(* IEC 61131-3 sources: POMIRTS_lab3/AS/Library_2/AsIORTI, 3 files *)

(* ---- AsIORTI.typ ---- *)
TYPE
	IORTI_DOUTTIME : 	STRUCT
		MODE_INACT : UDINT := 16#00000000; (*Digital Output Mode inactiv*)
		MODE_BOOL : UDINT := 16#00000001; (*Digital Output Mode boolean *)
		MODE_BASE_OFFS : UDINT := 16#00000002; (*Digital Output Mode Base and Offset one shot*)
		MODE_BASE_OFFS_PER : UDINT := 16#00000004; (*Digital Output Mode Base and Offset periodic*)
		MODE_ABSOLUT : UDINT := 16#00000008; (*Digital Output Mode absolut comparator values*)
		MODE_BOOL_INV : UDINT := 16#00000011; (*Digital Output Mode boolean inverted*)
		MODE_BASE_OFFS_INV : UDINT := 16#00000012; (*Digital Output Mode Base and Offset one shot  inverted*)
		MODE_BASE_OFFS_PER_INV : UDINT := 16#00000014; (*Digital Output Mode Base and Offset periodic  inverted*)
		MODE_ABSOLUT_INV : UDINT := 16#00000018; (*Digital Output Mode absolut comparator values inverted*)
	END_STRUCT;
	IORTI_COMP : 	STRUCT
		MODE_DISABLE : UDINT := 16#00000000; (*Comp Mode inactive*)
		MODE_ENABLE : UDINT := 16#00000001; (*Comp Mode active*)
		MODE_EQ : UDINT := 16#00000003; (*In1 is equal to In2*)
		MODE_NE : UDINT := 16#0000000D; (*In1 is not equal to In2*)
		MODE_GTU : UDINT := 16#00000005; (*In1 is greater than In2   (unsigned)*)
		MODE_GEU : UDINT := 16#00000007; (*In1 is greater or equal to In2   (unsigned)*)
		MODE_LTU : UDINT := 16#00000009; (*In1 is less than In2   (unsigned)*)
		MODE_LEU : UDINT := 16#0000000B; (*In1 is less or equal to In2   (unsigned)*)
		MODE_GT : UDINT := 16#80000005; (*In1 is greater than In2   (signed)*)
		MODE_GE : UDINT := 16#80000007; (*In1 is greater or equal to In2   (signed)*)
		MODE_LT : UDINT := 16#80000009; (*In1 is less than In2   (signed)*)
		MODE_LE : UDINT := 16#8000000B; (*In1 is less or equal to In2   (signed)*)
	END_STRUCT;
	IORTI_MUL : 	STRUCT
		MODE_UNSIGNED : UDINT := 16#00000000; (*Multiplication Mode unsigned*)
		MODE_SIGNED : UDINT := 16#80000000; (*Multiplication Mode signed*)
	END_STRUCT;
	IORTI_DIV : 	STRUCT
		MODE_UNSIGNED : UDINT := 16#00000000; (*Division Mode unsigned*)
		MODE_SIGNED : UDINT := 16#80000000; (*Division Mode signed*)
	END_STRUCT;
	IORTI_PWM : 	STRUCT
		MODE_INACT : UDINT := 16#00000000; (*Pwm Mode inactiv*)
		MODE_LEFT_PROC : UDINT := 16#00000001; (*Pwm Mode active left aligned  hightime as procentual value*)
		MODE_LEFT_PROC_DB : UDINT := 16#00000009; (*Pwm Mode active left aligned  hightime as procentual value, deadband enable*)
		MODE_LEFT_PROC_INV : UDINT := 16#00000011; (*Pwm Mode active left aligned  hightime as procentual value, inverted*)
		MODE_LEFT_PROC_DB_INV : UDINT := 16#00000019; (*Pwm Mode active left aligned  hightime as procentual value, deadband enable, inverted*)
		MODE_LEFT_TIME : UDINT := 16#00000005; (*Pwm Mode active left aligned  hightime as time value*)
		MODE_LEFT_TIME_DB : UDINT := 16#0000000D; (*Pwm Mode active left aligned  hightime as time value, deadband enable*)
		MODE_LEFT_TIME_INV : UDINT := 16#00000015; (*Pwm Mode active left aligned  hightime as time value, inverted*)
		MODE_LEFT_TIME_DB_INV : UDINT := 16#0000001D; (*Pwm Mode active left aligned  hightime as time value, deadband enable, inverted*)
		MODE_CENT_PROC : UDINT := 16#00000003; (*Pwm Mode active centered hightime as procentual value*)
		MODE_CENT_PROC_DB : UDINT := 16#0000000B; (*Pwm Mode active centered hightime as procentual value, deadband enable*)
		MODE_CENT_PROC_INV : UDINT := 16#00000013; (*Pwm Mode active centered hightime as procentual value, inverted*)
		MODE_CENT_PROC_DB_INV : UDINT := 16#0000001B; (*Pwm Mode active centered hightime as procentual value, deadband enable, inverted*)
		MODE_CENT_TIME : UDINT := 16#00000007; (*Pwm Mode active centered hightime as time value*)
		MODE_CENT_TIME_DB : UDINT := 16#0000000F; (*Pwm Mode active centered hightime as time value, deadband enable*)
		MODE_CENT_TIME_INV : UDINT := 16#00000017; (*Pwm Mode active centered hightime as time value, inverted*)
		MODE_CENT_TIME_DB_INV : UDINT := 16#0000001F; (*Pwm Mode active centered hightime as time value, deadband enable, inverted*)
		MODE_USE_START_AS_BASE : UDINT := 16#00000020; (*Pwm Mode Start used as Basetime*)
	END_STRUCT;
	IORTI_COUNT : 	STRUCT
		MODE_UPDWN_NOSTOP : UDINT := 16#00000000; (*Eventcounter Mode Up/Down with overrun*)
		MODE_CLKDIR_NOSTOP : UDINT := 16#00000001; (*Eventcounter Mode Clock and direction with overrun*)
		MODE_UPDWN_STOP : UDINT := 16#00000002; (*Eventcounter Mode Up/Down, stop at overrun*)
		MODE_CLKDIR_STOP : UDINT := 16#00000003; (*Eventcounter Mode Clock and direction, stop at overrun*)
	END_STRUCT;
	IORTI_REGISTER : 	STRUCT
		MODE_FREEZED : UDINT := 16#00000000; (*Register freezed*)
		MODE_TRANSPARENT : UDINT := 16#00000001; (*Register transparent*)
		MODE_EDGE_RISING : UDINT := 16#00000010; (*Register latch on rising edge*)
		MODE_EDGE_FALLING : UDINT := 16#00000011; (*Register latch on falling edge*)
		MODE_EDGE_BOTH : UDINT := 16#00000012; (*Register latch on both edges*)
		MODE_LEVEL_LOW : UDINT := 16#00000020; (*Register transparent if Latch low*)
		MODE_LEVEL_HIGH : UDINT := 16#00000021; (*Register transparent if Latch high*)
	END_STRUCT;
	IORTI_REAL : 	STRUCT
		TYPE_NORM : DINT := 16#00000000; (*Result is normalized*)
		TYPE_ZERO : DINT := 16#00000001; (*Result is zero*)
		TYPE_NAN : DINT := 16#00000002; (*Result is not a number*)
		TYPE_UNDER : DINT := 16#00000004; (*Result is underflow *)
		TYPE_OVER : DINT := 16#00000008; (*Result is overflow*)
		TYPE_DIVZERO : DINT := 16#00000010; (*Result is divide by zero*)
		TYPE_INFINITE : DINT := 16#00000020; (*Result is infinite*)
	END_STRUCT;
END_TYPE

(* ---- AsIORTI.fun ---- *)
FUNCTION_BLOCK rtiABCnt {ReActionFunctionNr 6}  {ReActionPhysical Channel} {ReActionPhysicalUnique ABR} (*AB Counter with latch*)
	VAR_INPUT
		Channel : INT;
		Mode : DINT;
		LatchEnable : DINT;
		LatchConfig : DINT;
		ForceOn : DINT;
		ForceCnt : DINT;
		ForceLatch : DINT;
		SimulCnt : {ReActionSimulParam} DINT;
		SimulLatch : {ReActionSimulParam} BOOL;
	END_VAR
	VAR_OUTPUT
		Cnt : DINT;
		CntTs : DINT;
		Latch : DINT;
		LatchTs : DINT;
		Status : DINT;
	END_VAR
	VAR
		LocLatch : DINT;
	END_VAR
END_FUNCTION_BLOCK

FUNCTION_BLOCK rtiABRPos {ReActionFunctionNr 7}  {ReActionPhysical Channel} {ReActionPhysicalUnique ABR} (*ABR Counter*)
	VAR_INPUT
		Channel : INT;
		Mode : DINT;
		RefEnable : DINT;
		RefConfig : DINT;
		RefPos : DINT;
		ForceOn : DINT;
		ForceVal : DINT;
		SimulPos : {ReActionSimulParam} DINT;
		SimulRef : {ReActionSimulParam} BOOL;
	END_VAR
	VAR_OUTPUT
		Pos : DINT;
		PosTs : DINT;
		Status : DINT;
	END_VAR
	VAR
		LocRefPos : DINT;
		LocRefDone : DINT;
		LocRefIn : BOOL;
	END_VAR
END_FUNCTION_BLOCK

FUNCTION_BLOCK rtiAbs {ReActionFunctionNr 121}		(*absolute value of signed value*)
	VAR_INPUT
		In : DINT;
	END_VAR
	VAR_OUTPUT
		Out : DINT;
	END_VAR
END_FUNCTION_BLOCK

FUNCTION_BLOCK rtiAdd {ReActionFunctionNr 107}		(*add In1 and In2*)
	VAR_INPUT
		In1 : DINT;
		In2 : DINT;
	END_VAR
	VAR_OUTPUT
		Out : DINT;
	END_VAR
END_FUNCTION_BLOCK

FUNCTION_BLOCK rtiAddSubReal {ReActionFunctionNr 130}	(*add or sub  In1 and In2*)
	VAR_INPUT
		In1 : REAL;
		In2 : REAL;
		Mode : DINT;
	END_VAR
	VAR_OUTPUT
		Out : REAL;
		Status : DINT;
	END_VAR
END_FUNCTION_BLOCK

FUNCTION_BLOCK rtiAin {ReActionFunctionNr 4}  {ReActionPhysical Channel} {ReActionPhysicalUnique}	(*read analog input channel*)
	VAR_INPUT
		Channel : INT;
		Filter : DINT;
		ForceOn : DINT;
		ForceVal : DINT;
		Simul : {ReActionSimulParam} DINT;
	END_VAR
	VAR_OUTPUT
		Out : DINT;
		Status : DINT;
	END_VAR
END_FUNCTION_BLOCK

FUNCTION_BLOCK rtiAnd {ReActionFunctionNr 100}	(*bitwise AND*)
	VAR_INPUT
		In1 : DINT;
		In2 : DINT;
		In3 : DINT;
		In4 : DINT;
	END_VAR
	VAR_OUTPUT
		OutTsEdge : DINT;
		Out : DINT;
		OutN : DINT;
	END_VAR
END_FUNCTION_BLOCK

FUNCTION_BLOCK rtiAnLimit {ReActionFunctionNr 118}	(*limit analog input value*)
	VAR_INPUT
		In : DINT;
		StatusIn : DINT;
		LowLimit : DINT;
		HighLimit : DINT;
	END_VAR
	VAR_OUTPUT
		Out : DINT;
		Status : DINT;
	END_VAR
END_FUNCTION_BLOCK

FUNCTION_BLOCK rtiAout {ReActionFunctionNr 5}  {ReActionPhysical Channel} {ReActionPhysicalUnique} (*write analog output channel*)
	VAR_INPUT
		Channel : INT;
		Enable : DINT;
		In : DINT;
		ForceOn : DINT;
		ForceVal : DINT;
	END_VAR
	VAR_OUTPUT
		OutRef : DINT;
		Simul : {ReActionSimulParam} DINT;
	END_VAR
END_FUNCTION_BLOCK

FUNCTION_BLOCK rtiBit2Byte {ReActionFunctionNr 119}	(*combines 8 bits into 1 byte*)
	VAR_INPUT
		In1 : DINT;
		In2 : DINT;
		In3 : DINT;
		In4 : DINT;
		In5 : DINT;
		In6 : DINT;
		In7 : DINT;
		In8 : DINT;
	END_VAR
	VAR_OUTPUT
		Out : DINT;
	END_VAR
END_FUNCTION_BLOCK

FUNCTION_BLOCK rtiByte2Bit {ReActionFunctionNr 120}	(*splits 1 byte into 8 bits*)
	VAR_INPUT
		In : DINT;
	END_VAR
	VAR_OUTPUT
		Out1 : DINT;
		Out2 : DINT;
		Out3 : DINT;
		Out4 : DINT;
		Out5 : DINT;
		Out6 : DINT;
		Out7 : DINT;
		Out8 : DINT;
	END_VAR
END_FUNCTION_BLOCK

FUNCTION_BLOCK rtiComp {ReActionFunctionNr 104}	(*compares In1 and In2 depending on the Mode*)
	VAR_INPUT
		Mode : UDINT;
		In1 : DINT;
		In2 : DINT;
	END_VAR
	VAR_OUTPUT
		StatusTsEdgePos : DINT;
		Status : DINT;
	END_VAR
END_FUNCTION_BLOCK

FUNCTION_BLOCK rtiCompReal {ReActionFunctionNr 133}	(*compares In1 and In2 depending on the Mode*)
	VAR_INPUT
		Mode : UDINT;
		In1 : REAL;
		In2 : REAL;
	END_VAR
	VAR_OUTPUT
		StatusTsEdgePos : DINT;
		Status : DINT;
		Result : DINT;
	END_VAR
END_FUNCTION_BLOCK

FUNCTION_BLOCK rtiCount {ReActionFunctionNr 115}	(*Up-Down counter or Clock-Direction counter, level sensitive*)
	VAR_INPUT
		Mode : UDINT;
		Up_Clk : DINT;
		Down_Dir : DINT;
		Clear : DINT;
	END_VAR
	VAR_OUTPUT
		OvlTsEdgePos : DINT;
		Out : DINT;
	END_VAR
END_FUNCTION_BLOCK

FUNCTION_BLOCK rtiDelay {ReActionFunctionNr 113}	(*delay signal for 1 reACTION cycle*)
	VAR_INPUT
		In : DINT;
	END_VAR
	VAR_OUTPUT
		Out : DINT;
		Out1 : DINT;
		Out2 : DINT;
		Out3 : DINT;
		Out4 : DINT;
	END_VAR
END_FUNCTION_BLOCK

FUNCTION_BLOCK rtiDelayReal {ReActionFunctionNr 113}	(*delay signal for 1 reACTION cycle*)
	VAR_INPUT
		In : REAL;
	END_VAR
	VAR_OUTPUT
		Out : REAL;
		Out1 : REAL;
		Out2 : REAL;
		Out3 : REAL;
		Out4 : REAL;
	END_VAR
END_FUNCTION_BLOCK

FUNCTION_BLOCK rtiDeMux {ReActionFunctionNr 117}	(*demultiplexer for 4 outputs*)
	VAR_INPUT
		Mux : DINT;
		In : DINT;
	END_VAR
	VAR_OUTPUT
		Out1 : DINT;
		Out2 : DINT;
		Out3 : DINT;
		Out4 : DINT;
	END_VAR
END_FUNCTION_BLOCK

FUNCTION_BLOCK rtiDeMuxReal {ReActionFunctionNr 117}	(*demultiplexer for 4 outputs*)
	VAR_INPUT
		Mux : DINT;
		In : REAL;
	END_VAR
	VAR_OUTPUT
		Out1 : REAL;
		Out2 : REAL;
		Out3 : REAL;
		Out4 : REAL;
	END_VAR
END_FUNCTION_BLOCK

FUNCTION_BLOCK rtiDin {ReActionFunctionNr 1} {ReActionPhysical Channel} {ReActionPhysicalUnique}	(*read digital input channel*)
	VAR_INPUT
		Channel : INT;
		Mode : UDINT;
		Filter : DINT;
		ForceOn : DINT;
		ForceVal : DINT;
		Simul : {ReActionSimulParam} BOOL;
	END_VAR
	VAR_OUTPUT
		OutTsEdgePos : DINT;
		OutTsEdgeNeg : DINT;
		Out : DINT;
	END_VAR
END_FUNCTION_BLOCK

FUNCTION_BLOCK rtiDiv {ReActionFunctionNr 110}	(*division*)
	VAR_INPUT
		Mode : UDINT;
		In1 : DINT;
		In2 : DINT;
	END_VAR
	VAR_OUTPUT
		Quotient : DINT;
		Remainder : DINT;
	END_VAR
END_FUNCTION_BLOCK

FUNCTION_BLOCK rtiDivReal {ReActionFunctionNr 132}	(*division*)
	VAR_INPUT
		In1 : REAL;
		In2 : REAL;
	END_VAR
	VAR_OUTPUT
		Quotient : REAL;
		Status : DINT;
	END_VAR
END_FUNCTION_BLOCK

FUNCTION_BLOCK rtiDout {ReActionFunctionNr 2} {ReActionPhysical Channel}  {ReActionPhysicalUnique DigitalOutputs}	(*write digital output channel*)
	VAR_INPUT
		Channel : INT;
		Enable : DINT;
		In : DINT;
		ForceOn : DINT;
		ForceVal : DINT;
	END_VAR
	VAR_OUTPUT
		Simul : {ReActionSimulParam} BOOL;
	END_VAR
END_FUNCTION_BLOCK

FUNCTION_BLOCK rtiDoutTime {ReActionFunctionNr 3} {ReActionPhysical Channel} {ReActionPhysicalUnique DigitalOutputs}	(*write digital output channel*)
	VAR_INPUT
		Channel : INT;
		Mode : UDINT;
		Comp1 : DINT;
		Comp2 : DINT;
		Base : DINT;
		Period : DINT;
		ForceOn : DINT;
		ForceVal : DINT;
	END_VAR
	VAR_OUTPUT
		EdgeCount : DINT;
		Simul : {ReActionSimulParam} BOOL;
	END_VAR
	VAR
		LocLatch : DINT;
		LocStat : DINT;
	END_VAR
END_FUNCTION_BLOCK

FUNCTION_BLOCK rtiIntToReal {ReActionFunctionNr 128}	 (*convert int to real with decimal point offset*)
	VAR_INPUT
		In : DINT;
		Shift : DINT;
	END_VAR
	VAR_OUTPUT
		Out : REAL;
		Status : DINT;
	END_VAR
END_FUNCTION_BLOCK

FUNCTION_BLOCK rtiInvertReal {ReActionFunctionNr 134}   (*invert input*)
	VAR_INPUT
		In : REAL;
	END_VAR
	VAR_OUTPUT
		Out : REAL;
		Status : DINT;
	END_VAR
END_FUNCTION_BLOCK

FUNCTION_BLOCK rtiLatch {ReActionFunctionNr 105}	(*latch value*)
	VAR_INPUT
		In : DINT;
		Latch : DINT;
	END_VAR
	VAR_OUTPUT
		Out : DINT;
	END_VAR
	VAR
		LocLatch : DINT;
	END_VAR
END_FUNCTION_BLOCK

FUNCTION_BLOCK rtiLatchReal {ReActionFunctionNr 105}	(*latch value*)
	VAR_INPUT
		In : REAL;
		Latch : DINT;
	END_VAR
	VAR_OUTPUT
		Out : REAL;
	END_VAR
END_FUNCTION_BLOCK

FUNCTION_BLOCK rtiMul {ReActionFunctionNr 109}	(*multiplication*)
	VAR_INPUT
		Mode : UDINT;
		In1 : DINT;
		In2 : DINT;
	END_VAR
	VAR_OUTPUT
		OutL : DINT;
		OutH : DINT;
	END_VAR
END_FUNCTION_BLOCK

FUNCTION_BLOCK rtiMulReal {ReActionFunctionNr 131}	(*multiplication*)
	VAR_INPUT
		In1 : REAL;
		In2 : REAL;
	END_VAR
	VAR_OUTPUT
		Out : REAL;
		Status : DINT;
	END_VAR
END_FUNCTION_BLOCK

FUNCTION_BLOCK rtiMux {ReActionFunctionNr 116}	(*select a value from 4 input values*)
	VAR_INPUT
		Mux : DINT;
		In1 : DINT;
		In2 : DINT;
		In3 : DINT;
		In4 : DINT;
	END_VAR
	VAR_OUTPUT
		Out : DINT;
	END_VAR
END_FUNCTION_BLOCK

FUNCTION_BLOCK rtiMuxReal {ReActionFunctionNr 116}	(*select a value from 4 input values*)
	VAR_INPUT
		Mux : DINT;
		In1 : REAL;
		In2 : REAL;
		In3 : REAL;
		In4 : REAL;
	END_VAR
	VAR_OUTPUT
		Out : REAL;
	END_VAR
END_FUNCTION_BLOCK

FUNCTION_BLOCK rtiNot {ReActionFunctionNr 103}	(*bitwise NOT*)
	VAR_INPUT
		In : DINT;
	END_VAR
	VAR_OUTPUT
		Out : DINT;
	END_VAR
END_FUNCTION_BLOCK

FUNCTION_BLOCK rtiOr {ReActionFunctionNr 101}	(*bitwise OR*)
	VAR_INPUT
		In1 : DINT;
		In2 : DINT;
		In3 : DINT;
		In4 : DINT;
	END_VAR
	VAR_OUTPUT
		OutTsEdge : DINT;
		Out : DINT;
		OutN : DINT;
	END_VAR
END_FUNCTION_BLOCK

FUNCTION_BLOCK rtiPar {ReActionPhysical DpNr}	(*read parameter from cyclic datapoint*)
	VAR_INPUT
		DpNr : INT;
		Simul : {ReActionSimulParam} DINT;
	END_VAR
	VAR_OUTPUT
		Data : DINT;
	END_VAR
END_FUNCTION_BLOCK

FUNCTION_BLOCK rtiParReal {ReActionPhysical DpNr}	 (*read parameter from cyclic datapoint*)
	VAR_INPUT
		DpNr : INT;
		Simul : {ReActionSimulParam} REAL;
	END_VAR
	VAR_OUTPUT
		Data : REAL;
	END_VAR
END_FUNCTION_BLOCK

FUNCTION_BLOCK rtiPwm {ReActionFunctionNr 114}	(*generate PWM signal, must be followed by rtiDoutTime*)
	VAR_INPUT
		Mode : UDINT;
		Start : DINT;
		Period : DINT;
		Duty : DINT;
		DeadB : DINT;
	END_VAR
	VAR_OUTPUT
		ModeOut : UDINT;
		OutTsEdgePos : DINT;
		OutTsEdgeNeg : DINT;
		Base : DINT;
		PeriodOut : DINT;
	END_VAR
END_FUNCTION_BLOCK

FUNCTION_BLOCK rtiRealToInt  {ReActionFunctionNr 129}  (*convert real to int with decimal point offset*)
	VAR_INPUT
		In : REAL;
		Shift : DINT;
	END_VAR
	VAR_OUTPUT
		Out : DINT;
		Status : DINT;
	END_VAR
END_FUNCTION_BLOCK

FUNCTION_BLOCK rtiRegister  {ReActionFunctionNr 124} (*register values*)
	VAR_INPUT
		Mode : UDINT;
		Latch : DINT;
		In1 : DINT;
		In2 : DINT;
		In3 : DINT;
		In4 : DINT;
	END_VAR
	VAR_OUTPUT
		OutTsLatch : DINT;
		Out1 : DINT;
		Out2 : DINT;
		Out3 : DINT;
		Out4 : DINT;
	END_VAR
	VAR
		LocLatch : DINT;
	END_VAR
END_FUNCTION_BLOCK

FUNCTION_BLOCK rtiRegisterReal  {ReActionFunctionNr 124} (*register values*)
	VAR_INPUT
		Mode : UDINT;
		Latch : DINT;
		In1 : REAL;
		In2 : REAL;
		In3 : REAL;
		In4 : REAL;
	END_VAR
	VAR_OUTPUT
		OutTsLatch : DINT;
		Out1 : REAL;
		Out2 : REAL;
		Out3 : REAL;
		Out4 : REAL;
	END_VAR
	VAR
		LocLatch : DINT;
	END_VAR
END_FUNCTION_BLOCK

FUNCTION_BLOCK rtiRes {ReActionPhysical DpNr}  {ReActionPhysicalUnique Results}	(*write results to cyclic datapoint*)
	VAR_INPUT
		DpNr : INT;
		Data : DINT;
	END_VAR
	VAR_OUTPUT
		Simul : {ReActionSimulParam} DINT;
	END_VAR
END_FUNCTION_BLOCK

FUNCTION_BLOCK rtiResReal {ReActionPhysical DpNr}  {ReActionPhysicalUnique Results}	(*write results to cyclic datapoint*)
	VAR_INPUT
		DpNr : INT;
		Data : REAL;
	END_VAR
	VAR_OUTPUT
		Simul : {ReActionSimulParam} REAL;
	END_VAR
END_FUNCTION_BLOCK

FUNCTION_BLOCK rtiRF_TRIG {ReActionFunctionNr 122}	(*detect rising/falling edge of input signal*)
	VAR_INPUT
		CLK : DINT;
	END_VAR
	VAR_OUTPUT
		OutEdge : DINT;
		OutEdgePos : DINT;
		OutEdgeNeg : DINT;
	END_VAR
	VAR
		LocLatch : DINT;
	END_VAR
END_FUNCTION_BLOCK

FUNCTION_BLOCK rtiShift {ReActionFunctionNr 111}	(*arithmetic or logigal shift*)
	VAR_INPUT
		In : DINT;
		Shl : DINT;
		Shr : DINT;
	END_VAR
	VAR_OUTPUT
		Out : DINT;
	END_VAR
END_FUNCTION_BLOCK

FUNCTION_BLOCK rtiSineReal {ReActionFunctionNr 136} (*sine*)
	VAR_INPUT
		In : REAL;
	END_VAR
	VAR_OUTPUT
		Out : REAL;
		Status : DINT;
	END_VAR
END_FUNCTION_BLOCK

FUNCTION_BLOCK rtiSqrtReal {ReActionFunctionNr 135}	(*square root*)
	VAR_INPUT
		In : REAL;
	END_VAR
	VAR_OUTPUT
		Out : REAL;
		Status : DINT;
	END_VAR
END_FUNCTION_BLOCK

FUNCTION_BLOCK rtiSRff {ReActionFunctionNr 106}	(*SR flipflop*)
	VAR_INPUT
		InS : DINT;
		InR : DINT;
	END_VAR
	VAR_OUTPUT
		OutTsEdge : DINT;
		Out : DINT;
	END_VAR
END_FUNCTION_BLOCK

FUNCTION_BLOCK rtiSSI {ReActionFunctionNr 8}  {ReActionPhysical Channel} {ReActionPhysicalUnique} (*SSI Encoder*)
	VAR_INPUT
		Channel : INT;
		Mode : DINT;
		Trigger : DINT;
		ForceOn : DINT;
		ForceVal : DINT;
		SimulPos : {ReActionSimulParam} DINT;
	END_VAR
	VAR_OUTPUT
		Pos : DINT;
		PosTs : DINT;
		Status : DINT;
	END_VAR
END_FUNCTION_BLOCK

FUNCTION_BLOCK rtiSub {ReActionFunctionNr 108}	(*subtraction*)
	VAR_INPUT
		In1 : DINT;
		In2 : DINT;
	END_VAR
	VAR_OUTPUT
		Out : DINT;
	END_VAR
END_FUNCTION_BLOCK

FUNCTION_BLOCK rtiTDel {ReActionFunctionNr 112}	(*compare time delays*)
	VAR_INPUT
		Enable : DINT;
		Comp1 : DINT;
		Comp2 : DINT;
		Comp3 : DINT;
		Comp4 : DINT;
		Comp5 : DINT;
		Comp6 : DINT;
		Base : DINT;
	END_VAR
	VAR_OUTPUT
		Out : DINT;
	END_VAR
	VAR
		LocStat : DINT;
	END_VAR
END_FUNCTION_BLOCK

FUNCTION_BLOCK rtiTime {ReActionFunctionNr 252}	(*get time of cycle start and last parameter refresh*)
	VAR_OUTPUT
		TsPar : DINT;
		TsCycle : DINT;
	END_VAR
END_FUNCTION_BLOCK

FUNCTION_BLOCK rtiTimeLoc2Net {ReActionFunctionNr 250}	(*converts local time [10ns] to NetTime [1/256us]*)
	VAR_INPUT
		LocTime : DINT;
	END_VAR
	VAR_OUTPUT
		NetTime : DINT;
	END_VAR
END_FUNCTION_BLOCK

FUNCTION_BLOCK rtiTimeNet2Loc {ReActionFunctionNr 251}	(*converts NetTime [1/256us] to local time [10ns]*)
	VAR_INPUT
		NetTime : DINT;
	END_VAR
	VAR_OUTPUT
		LocTime : DINT;
	END_VAR
END_FUNCTION_BLOCK

FUNCTION_BLOCK rtiTP {ReActionFunctionNr 123}	(*generates TRUE-pulse on rising edge of input signal*)
	VAR_INPUT
		IN : DINT;
		PT : DINT;
	END_VAR
	VAR_OUTPUT
		Q : DINT;
		ET : DINT;
	END_VAR
	VAR
		LocLatch : DINT;
	END_VAR
END_FUNCTION_BLOCK

FUNCTION_BLOCK rtiVarRead {ReActionPhysical DpNr}	(*reads from internal variable*)
	VAR_INPUT
		DpNr : INT;
		Simul : {ReActionSimulParam} DINT;
	END_VAR
	VAR_OUTPUT
		Out : DINT;
	END_VAR
END_FUNCTION_BLOCK

FUNCTION_BLOCK rtiVarReadReal {ReActionPhysical DpNr}	(*reads from internal variable*)
	VAR_INPUT
		DpNr : INT;
		Simul : {ReActionSimulParam} REAL;
	END_VAR
	VAR_OUTPUT
		Out : REAL;
	END_VAR
END_FUNCTION_BLOCK

FUNCTION_BLOCK rtiVarWrite {ReActionPhysical DpNr}  {ReActionPhysicalUnique VarWrite}	(*writes to internal variable*)
	VAR_INPUT
		DpNr : INT;
		In : DINT;
	END_VAR
	VAR_OUTPUT
		Simul : {ReActionSimulParam} DINT;
	END_VAR
END_FUNCTION_BLOCK

FUNCTION_BLOCK rtiVarWriteReal {ReActionPhysical DpNr}  {ReActionPhysicalUnique VarWrite}	(*writes to internal variable*)
	VAR_INPUT
		DpNr : INT;
		In : REAL;
	END_VAR
	VAR_OUTPUT
		Simul : {ReActionSimulParam} REAL;
	END_VAR
END_FUNCTION_BLOCK

FUNCTION_BLOCK rtiXor {ReActionFunctionNr 102}	(*bitwise XOR*)
	VAR_INPUT
		In1 : DINT;
		In2 : DINT;
		In3 : DINT;
		In4 : DINT;
	END_VAR
	VAR_OUTPUT
		OutTsEdge : DINT;
		Out : DINT;
		OutN : DINT;
	END_VAR
END_FUNCTION_BLOCK

FUNCTION_BLOCK rtiSim (*control simulation mode (no effect on reACTION IO module)*)
	VAR_INPUT
		Enable : {ReActionSimulParam} BOOL;
		Mode : {ReActionSimulParam} UDINT;
		Clear : {ReActionSimulParam} BOOL;
	END_VAR
	VAR_OUTPUT
		Cycles : {ReActionSimulParam} UDINT;
		Status : {ReActionSimulParam} UINT;
	END_VAR
END_FUNCTION_BLOCK

(* ---- AsIORTI.var ---- *)
VAR CONSTANT
	IORTI_SIM_MODE_DEFAULT : UDINT := 16#00000001; (* Default simulation mode *)
	IORTI_SIM_ERR_UNKNOWN_MODE : UDINT := 37910; (* unknown simulation mode selected *)
	IORTI_SIM_ERR_OUT_OF_MEMORY : UDINT := 37911; (* out of memory error *)
	IORTI_SIM_ERR_INVALID_DPNR : UDINT := 37912; (* invalid datapoint number *)
	IORTI_SIM_ERR_PAR_SIMUL_VALUE : UDINT := 37913; (* simulation values for parameters with the same DpNr are not equal *)
	IORTI_SIM_ERR_VAR_SIMUL_VALUE : UDINT := 37914; (* simulation values for variables with the same DpNr are not equal *)
END_VAR
